(* IEC 61131-3 sources: CodesysTest/export/Function Blocks/FB_InternalLogger.pou, 2 files *)

(* ---- FB_InternalLogger.pou.st ---- *)
(*#-#-#-#-#-#-#-#-#-#---Declaration---#-#-#-#-#-#-#-#-#-#-#-#-#*)

FUNCTION_BLOCK FB_InternalLogger IMPLEMENTS IMachineLogger
VAR_INPUT
END_VAR
VAR_OUTPUT
END_VAR
VAR
	//loggedItems : ARRAY[0..500] OF FaultLogType;
	loggedItems : ARRAY[0..GlobalData.MAX_LOGGED_ITEMS] OF LogMessageType;
	numOfLogEntries : UINT;
	logFull : BOOL;
	RTC : FB_GetTime();
	clearLog : BOOL;
	i : UINT;
END_VAR
(*#-#-#-#-#-#-#-#-#-#---Implementation---#-#-#-#-#-#-#-#-#-#-#-#-#*)

//	Function Block: FB_Logger
//	Description: This is an internal logger for reference within Codesys.  It is an array that can be displayed on the TargetVisu/WebVisu
//
//	Created by: Ben Hess
//	Created Date: Tuesday, September 11, 2018

// DISABLED LOGGING FOR CREVIS PLC - SCAN TIMES OUT OF CONTROL

(* ---- AddLogItem.m.st ---- *)
(*#-#-#-#-#-#-#-#-#-#---Declaration---#-#-#-#-#-#-#-#-#-#-#-#-#*)

METHOD AddLogItem
VAR_INPUT
	//category : STRING;
	message : STRING;
END_VAR
(*#-#-#-#-#-#-#-#-#-#---Implementation---#-#-#-#-#-#-#-#-#-#-#-#-#*)
